// TIA Portal project "11062025" (V19)

(* hardware
DEVICE "S7-300/ET200M station_1"  S7-300 station
   slot 0: "Rail_0"  Rail  6ES7 390-1***0-0AA0
   slot 2: "PLC_1"  CPU 314C-2 PN/DP  6ES7 314-6EH04-0AB0  V3.3.18
      slot 2: "PROFINET interface_1"  PN-IO
         slot 1: "Port_1"  Port
         slot 2: "Port_2"  Port
      slot 5: "DI 24/DO 16_1"  DI24/DO16
      slot 6: "AI 5/AO 2_1"  AI5/AO2
      slot 7: "Count_1"  Counter
      slot 8: "Positioning_1"  Positioning
*)

// ===== PLC "PLC_1"  CPU 314C-2 PN/DP =====

VAR_GLOBAL   // PLC tag table "Default tag table"
   "Start Button 0" AT %I0.0 : Bool;
   "Stop Button 0" AT %I0.1 : Bool;
   "retroflective Sensor 0" AT %I0.2 : Bool;
   "off2" AT %I0.3 : Bool;
   "metal2" AT %I0.4 : Bool;
   "off1" AT %I0.5 : Bool;
   "retroflective sensor 1" AT %I0.6 : Bool;
   "atuador1" AT %Q0.0 : Bool;
   "atuador2" AT %Q0.1 : Bool;
   "motor1" AT %Q0.2 : Bool;
   "motor2" AT %Q0.3 : Bool;
   "motor esteira" AT %Q0.4 : Bool;
   "motor esteira2" AT %Q0.5 : Bool;
   "cap.initi" AT %I0.7 : Bool;
   "Tag_1" AT %I1.0 : Bool;
END_VAR

DATA_BLOCK "Block_1_DB"   // DB1
{ S7_Optimized_Access := 'FALSE' }
VERSION : 0.1
// stored: InstanceOfName Block_1
"Block_1"
BEGIN
END_DATA_BLOCK

DATA_BLOCK "Block_1_DB_1"   // DB2
{ S7_Optimized_Access := 'FALSE' }
VERSION : 0.1
// stored: InstanceOfName Block_1
"Block_1"
BEGIN
END_DATA_BLOCK

DATA_BLOCK "Block_1_DB_3"   // DB3
{ S7_Optimized_Access := 'FALSE' }
VERSION : 0.1
// stored: InstanceOfName Block_1
"Block_1"
BEGIN
END_DATA_BLOCK

DATA_BLOCK "Block_1_DB_2"   // DB5
{ S7_Optimized_Access := 'FALSE' }
VERSION : 0.1
// stored: InstanceOfName Block_1
"Block_1"
BEGIN
END_DATA_BLOCK

DATA_BLOCK "Block_1_DB_4"   // DB6
{ S7_Optimized_Access := 'FALSE' }
VERSION : 0.1
// stored: InstanceOfName Block_1
"Block_1"
BEGIN
END_DATA_BLOCK

FUNCTION_BLOCK "Block_1"   // FB1, SCL
{ S7_Optimized_Access := 'FALSE' }
VERSION : 0.1
   VAR_INPUT
      retroflecrive1 : Bool;
      off2 : Bool;
      metal2 : Bool;
      off1 : Bool;
      "retroflecrive 2" : Bool;
      "cap.initi" : Bool;
   END_VAR
   VAR_OUTPUT
      atuador1 : Bool;
      atuador2 : Bool;
      motor1 : Bool;
      motor2 : Bool;
      "motor esteira" : Bool;
      "motor esteira2" : Bool;
   END_VAR
   VAR
      memoria1 : Bool;
      memoria2 : Bool;
      memoria3 : Bool;
   END_VAR
BEGIN
   IF #"cap.initi" = 1 THEN
       #"motor esteira" := 1;
       #"motor esteira2" := 1;

   END_IF;


   IF #metal2 = 1 THEN
       #memoria1 := 1;
   END_IF;

   "IEC_Timer_0_DB".TON(IN := #memoria1,
                        PT := t#4s,
                        Q => #atuador2);
   IF #"off2" = 1 THEN
       #atuador1 := 0;
       #motor2 := 0;
   END_IF;

   IF #retroflecrive1 = 0 AND #"retroflecrive 2" = 0 THEN
       #atuador1 := 1;
       #motor2 := 1;
   END_IF;

   IF #"off1" = 1 THEN
       #atuador1 := 0;
       #motor2 := 0;
   END_IF;
END_FUNCTION_BLOCK

ORGANIZATION_BLOCK "Main"   // OB1, LAD
TITLE = "Main Program Sweep (Cycle)"
{ S7_Optimized_Access := 'FALSE' }
VERSION : 0.1
   VAR_TEMP
      OB1_EV_CLASS : Byte;   // Bits 0-3 = 1 (Coming event), Bits 4-7 = 1 (Event class 1)
      OB1_SCAN_1 : Byte;   // 1 (Cold restart scan 1 of OB 1), 3 (Scan 2-n of OB 1)
      OB1_PRIORITY : Byte;   // Priority of OB Execution
      OB1_OB_NUMBR : Byte;   // 1 (Organization block 1, OB1)
      OB1_RESERVED_1 : Byte;   // Reserved for system
      OB1_RESERVED_2 : Byte;   // Reserved for system
      OB1_PREV_CYCLE : Int;   // Cycle time of previous OB1 scan (milliseconds)
      OB1_MIN_CYCLE : Int;   // Minimum cycle time of OB1 (milliseconds)
      OB1_MAX_CYCLE : Int;   // Maximum cycle time of OB1 (milliseconds)
      OB1_DATE_TIME : Date_And_Time;   // Date and time OB1 started
   END_VAR
BEGIN

REGION Network 1
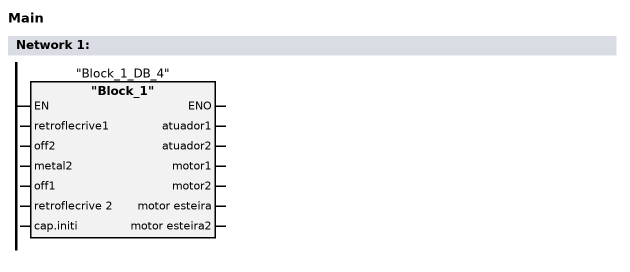
   RUNG wire#powerrail
      "Block_1_DB_4"(retroflecrive1 :=, off2 :=, metal2 :=, off1 :=, "retroflecrive 2" :=, "cap.initi" :=, atuador1 =>, atuador2 =>, motor1 =>, motor2 =>, "motor esteira" =>, "motor esteira2" =>)
   END_RUNG
   // the same network as SCL:
   "Block_1_DB_4"();   // "Block_1"
END_REGION
END_ORGANIZATION_BLOCK